FUNCTION f_MessageSet : BOOL
VAR_INPUT
  stMessage     : ST_Message;
END_VAR
VAR
  _uiIndex      : UINT;
  _MainDevice   : e_Device;
  _nModRes      : UDINT;     // residual after modulo
END_VAR

stMessage.tTime                     := GVL_MSG_XTS.sLocalTime;

// why here? so all calls to this function may stay the same
_nModRes                            := stMessage.eDevice MOD e_Device.General;
_MainDevice                         := stMessage.eDevice - _nModRes;

CASE _MainDevice
OF
  //--------------------------------------------------------------------------------
  e_device.DataProduct:
    // this is your data, if you choose to use this message system
    FOR _uiIndex := 1 TO GVL_MSG_XTS.MAX_MESSAGE
    DO
      IF (GVL_MSG_XTS.ProductMessages[_uiIndex].eType = e_MessageType.eMessageEmpty)
      THEN
        GVL_MSG_XTS.ProductMessages[_uiIndex]      := stMessage;
        GVL_MSG_XTS.MessageProductIndex            := _uiIndex;
        EXIT;
      END_IF
    END_FOR
  
    IF (stMessage.eType = E_MessageType.eMessageError)
    THEN
      // in case of error: increment counter
      GVL_MSG_XTS.MessageProductError              := GVL_MSG_XTS.MessageProductError + 1;
    END_IF
  //--------------------------------------------------------------------------------
  e_Device.Process,
  e_Device.Application:
    FOR _uiIndex := 1 TO GVL_MSG_XTS.MAX_MESSAGE
    DO
      IF (GVL_MSG_XTS.ApplicationMessages[_uiIndex].eType = e_MessageType.eMessageEmpty)
      THEN
        GVL_MSG_XTS.ApplicationMessages[_uiIndex]  := stMessage;    // yes, we grab global values directly, only here
        GVL_MSG_XTS.MessageApplicationIndex        := _uiIndex;
        EXIT;
      END_IF
    END_FOR
    IF (stMessage.eType = E_MessageType.eMessageError)
    THEN
      // in case of error: increment counter
      GVL_MSG_XTS.MessageApplicationError          := GVL_MSG_XTS.MessageApplicationError + 1;
    END_IF
  //--------------------------------------------------------------------------------
  e_Device.MetricsXts:
    FOR _uiIndex := 1 TO GVL_MSG_XTS.MAX_MESSAGE
    DO
      IF (GVL_MSG_XTS.MetricsMessages[_uiIndex].eType = e_MessageType.eMessageEmpty)
      THEN
        GVL_MSG_XTS.MetricsMessages[_uiIndex]      := stMessage;    // yes, we grab global values directly, only here
        GVL_MSG_XTS.MessageMetricsIndex            := _uiIndex;
        EXIT;
      END_IF
    END_FOR
    IF (stMessage.eType = E_MessageType.eMessageError)
    THEN
      // in case of error: increment counter
      GVL_MSG_XTS.MessageMetricsError              := GVL_MSG_XTS.MessageMetricsError + 1;
    END_IF
  //--------------------------------------------------------------------------------
  e_Device.MetricsAxis:
    FOR _uiIndex := 1 TO GVL_MSG_XTS.MAX_MESSAGE
    DO
      IF (GVL_MSG_AXIS.MetricMessages[_uiIndex].eType = e_MessageType.eMessageEmpty)
      THEN
        GVL_MSG_AXIS.MetricMessages[_uiIndex]  := stMessage;    // yes, we grab global values directly, only here
        GVL_MSG_AXIS.MessageMetricIndex        := _uiIndex;
        EXIT;
      END_IF
    END_FOR
    IF (stMessage.eType = E_MessageType.eMessageError)
    THEN
      // in case of error: increment counter
      GVL_MSG_AXIS.MessageMetricError          := GVL_MSG_AXIS.MessageMetricError + 1;
    END_IF
  //--------------------------------------------------------------------------------
  e_Device.Axis,
  e_Device.XfcAxis,
  e_device.XfcTouchProbe,
  e_device.XfcTriggerBox,
  e_Device.Camming,
  e_device.NciChannel,
  e_device.NciChannelCtrl:
    FOR _uiIndex := 1 TO GVL_MSG_XTS.MAX_MESSAGE
    DO
      IF (GVL_MSG_AXIS.MotionMessages[_uiIndex].eType = e_MessageType.eMessageEmpty)
      THEN
        GVL_MSG_AXIS.MotionMessages[_uiIndex]  := stMessage;    // yes, we grab global values directly, only here
        GVL_MSG_AXIS.MessageMotionIndex        := _uiIndex;
        EXIT;
      END_IF
    END_FOR
    IF (stMessage.eType = E_MessageType.eMessageError)
    THEN
      // in case of error: increment counter
      GVL_MSG_AXIS.MessageMotionError           := GVL_MSG_AXIS.MessageMotionError + 1;
    END_IF
  //--------------------------------------------------------------------------------
ELSE
  CASE stMessage.eDevice
  OF
    Device_MainApplication,
    Device_XmlData,              
    Device_Utilities:
      FOR _uiIndex := 1 TO GVL_MSG_XTS.MAX_MESSAGE
      DO
        IF (GVL_MSG_XTS.ApplicationMessages[_uiIndex].eType = e_MessageType.eMessageEmpty)
        THEN
          GVL_MSG_XTS.ApplicationMessages[_uiIndex]:= stMessage;    // yes, we grab global values directly, only here
          GVL_MSG_XTS.MessageApplicationIndex      := _uiIndex;
          EXIT;
        END_IF
      END_FOR
      IF (stMessage.eType = E_MessageType.eMessageError)
      THEN
        // in case of error: increment counter
        GVL_MSG_XTS.MessageApplicationError        := GVL_MSG_XTS.MessageApplicationError + 1;
      END_IF

    Device_MainAxis,
    Device_Nci,
    Device_Cam,
    Device_Functions,
    Device_FlyingSaw,
    Device_ParameterSelector:     // PLC_MOTION
      FOR _uiIndex := 1 TO GVL_MSG_XTS.MAX_MESSAGE
      DO
        IF (GVL_MSG_AXIS.MotionMessages[_uiIndex].eType = e_MessageType.eMessageEmpty)
        THEN
          GVL_MSG_AXIS.MotionMessages[_uiIndex]:= stMessage;    // yes, we grab global values directly, only here
          GVL_MSG_AXIS.MessageMotionIndex      := _uiIndex;
          EXIT;
        END_IF
      END_FOR
      IF (stMessage.eType = E_MessageType.eMessageError)
      THEN
        // in case of error: increment counter
        GVL_MSG_AXIS.MessageMotionError        := GVL_MSG_AXIS.MessageMotionError + 1;
      END_IF

    Device_Main,
    Device_MoverSelector:
      FOR _uiIndex := 1 TO GVL_MSG_XTS.MAX_MESSAGE
      DO
        IF (GVL_MSG_XTS.TransportMessages[_uiIndex].eType = e_MessageType.eMessageEmpty)
        THEN
          GVL_MSG_XTS.TransportMessages[_uiIndex]  := stMessage;
          GVL_MSG_XTS.MessageTransportIndex        := _uiIndex;
          EXIT;
        END_IF
      END_FOR
  ELSE    
    //--------------------------------------------------------------------------------
    FOR _uiIndex := 1 TO GVL_MSG_XTS.MAX_MESSAGE
    DO
      IF (GVL_MSG_XTS.TransportMessages[_uiIndex].eType = e_MessageType.eMessageEmpty)
      THEN
        GVL_MSG_XTS.TransportMessages[_uiIndex]    := stMessage;
        GVL_MSG_XTS.MessageTransportIndex          := _uiIndex;
        EXIT;
      END_IF
    END_FOR
  
    IF (stMessage.eType = E_MessageType.eMessageError)
    THEN
      // in case of error: increment counter
      GVL_MSG_XTS.MessageTransportError := GVL_MSG_XTS.MessageTransportError + 1;
    END_IF
  END_CASE
END_CASE

END_FUNCTION

(* stored: Version 1.1.0.1, ProductVersion 3.1.4026.18
   POU f_MessageSet: Id {b3f088c0-23db-44a1-a50a-6faad1d308c8}, SpecialFunc None *)
